// TIA Portal V16 export
// export: Created 2024-05-13T12:49:09.6013961Z, ExportSetting WithDefaults, DisplayName Totally Integrated Automation Portal, DisplayVersion V16 Update 6, DisplayName TIA Portal Version Control Interface, DisplayVersion V16 Update 2, DisplayName TIA Portal Openness, DisplayVersion V16 Update 6, DisplayName TIA Portal Test Suite Advanced, DisplayVersion V16, DisplayName SINAMICS Startdrive Advanced, DisplayVersion V16 Update 5, DisplayName SINAMICS Startdrive G130, G150, S120, S150, SINAMICS MV, S210, DisplayVersion V16 Update 5, DisplayName SINAMICS Startdrive G110M, G120, G120C, G120D, G120P, G115D, DisplayVersion V16 Update 5, DisplayName STEP 7 Professional, DisplayVersion V16 Update 6, DisplayName STEP 7 Safety, DisplayVersion V16, DisplayName WinCC Advanced, DisplayVersion V16 Update 6
TYPE "SCA_rotatingRollers_IO"
// stored: IsFailsafeCompliant false
   STRUCT
      Lifting_safety_switch_entry : Bool;   // Safety switch entry side
      Lifting_safety_switch_exit : Bool;   // Safety switch exit side
      Entry_up : Bool;   // Entry side up
      Entry_down : Bool;   // Entry side down
      Exit_up : Bool;   // Exit side up
      Exit_down : Bool;   // Exit side down
      Rotating_safety_switch : Bool;   // Safety switch rotating
      Entry_Side_Circuit_Braker : Bool;   // Entry Side Circuit Braker
      Exit_Side_Circuit_Braker : Bool;   // Exit Side Circuit Braker
      Man_rollers_up : Bool;   // Manual rollers up
      Man_rollers_down : Bool;   // Manual rollers down
      Man_cnv_fwd : Bool;   // Manual rollers fwd
      Man_cnv_rev : Bool;   // Manual rollers rev
   END_STRUCT;
END_TYPE
